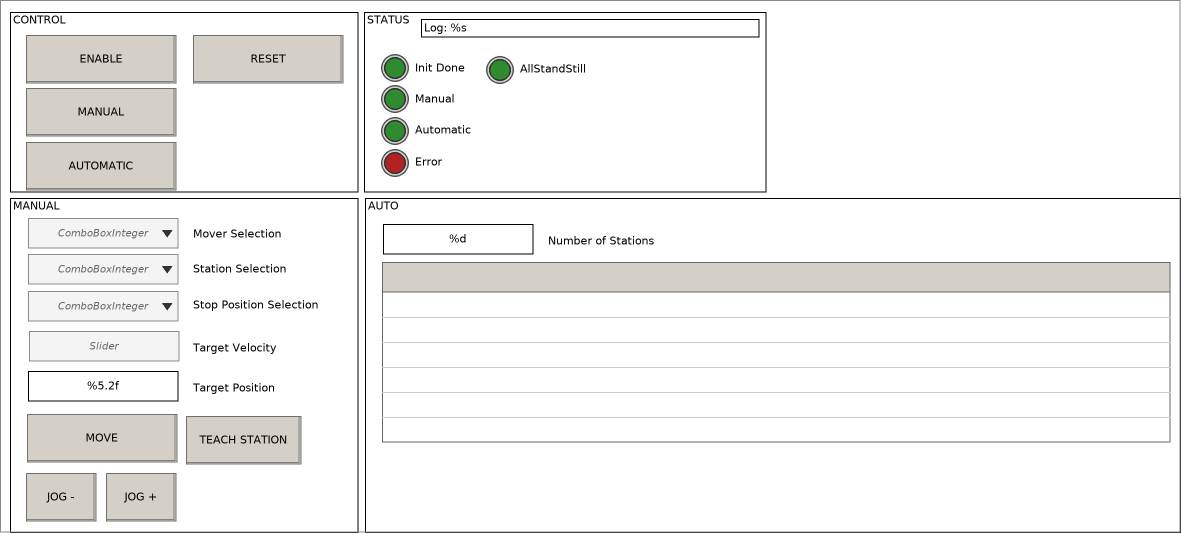
VISUALIZATION XTS_System_VISU  // 1181x533
VAR_IN_OUT
	xts : XTS_System;
END_VAR
    Rectangle (364,12 402x180), "STATUS"
    Rectangle (10,12 348x180), "CONTROL"
    Rectangle (10,198 348x335), "MANUAL"
    Button (26,35 150x48), "ENABLE"
        toggle xts.bEnable
    Button (26,88 150x48), "MANUAL"
        toggle xts.bManual
    Button (26,142 150x48), "AUTOMATIC"
        toggle xts.bAutomatic
    Lamp1 (379,52 32x32), variable: xts.bInitDone, style: Lamp-Lamp1-Green
    Label (412,53 110x30), "Init Done"
    ComboBoxInteger (28,218 150x30), variable: xts.udiMoverSelection
    ComboBoxInteger (28,254 150x30), variable: xts.udiStationSelection
    Label (190,219 150x30), "Mover Selection"
    Label (190,254 150x30), "Station Selection"
    ComboBoxInteger (28,291 150x30), variable: xts.udiStopPositionSelection
    Label (190,290 150x30), "Stop Position Selection"
    Button (27,414 150x48), "MOVE"
        tap xts.bManualMove
    Button (26,473 70x48), "JOG -"
        tap xts.bJogBackwards
    Button (106,473 70x48), "JOG +"
        tap xts.bJogForward
    Lamp1 (379,83 32x32), variable: xts.bInManual, style: Lamp-Lamp1-Green
    Label (412,84 110x30), "Manual"
    Lamp1 (379,115 32x32), variable: xts.bInAutomatic, style: Lamp-Lamp1-Green
    Label (412,115 110x30), "Automatic"
    Slider (29,331 150x30), variable: xts.lrTargetVelocity, scale 1..4000
    Label (190,333 150x30), "Target Velocity"
    Rectangle (28,371 150x30), "%5.2f", text variable: xts.lrTargetPosition
        OnMouseClick: write the text variable via Default
    Label (190,373 150x30), "Target Position"
    Button (186,416 115x48), "TEACH STATION"
        tap xts.bTeachStation
    Lamp1 (379,147 32x32), variable: xts.bError, style: Lamp-Lamp1-Red
    Label (412,147 110x30), "Error"
    Button (193,35 150x48), "RESET"
        tap xts.bReset
    Rectangle (365,198 816x335), "AUTO"
    Rectangle (383,224 150x30), "%d", text variable: xts.stCfg.udiNumStations
        OnMouseClick: write the text variable via Default
    Label (545,226 150x30), "Number of Stations"
    Table (382,262 788x180), data array: xts.stVisuStationsCfg
        p3854506369: xts.stVisuStationsCfg[INDEX].sName
        p1892666644: xts.stVisuStationsCfg[INDEX].lrStartPosition
        p338671338: xts.stVisuStationsCfg[INDEX].lrEndPosition
        p2170511999: xts.stVisuStationsCfg[INDEX].lrStopPosition
        p3723444502: xts.stVisuStationsCfg[INDEX].lrProcessingTime
        p1218418051: xts.stVisuStationsCfg[INDEX].uiNumStopPositions
        p746581629: xts.stVisuStationsCfg[INDEX].lrTravelTime
        p511219082: Start Position
        p1755163831: End Position
        p4092479075: Stop Position
        p2237128397: Processing Time
        p505689113: Num Stop Positions
        p1757482276: Travel Time
    Rectangle (421,19 338x18), "Log: %s", text variable: xts.sLog
        OnMouseClick: write the text variable via Default
    Lamp1 (484,54 32x32), variable: xts.bAllMoversStandStill, style: Lamp-Lamp1-Green
    Label (517,54 110x30), "AllStandStill"
END_VISUALIZATION

(* stored: Version 1.1.0.1, ProductVersion 3.1.4024.11
   Visu XTS_System_VISU: Id {1b0b2335-e4a4-4979-b98e-4146a6229b4a} *)
